FUNCTION TryConvert_BYTE_TO_WORD : BOOL
VAR_INPUT
	in : BYTE;
	out : REFERENCE TO WORD;
END_VAR

out := BYTE_TO_WORD(in);
TryConvert_BYTE_TO_WORD := TRUE;

END_FUNCTION

(* stored: Version 1.1.0.1, ProductVersion 3.1.4024.12
   POU TryConvert_BYTE_TO_WORD: Id {f96b26b8-9bd6-494d-887e-55a472e0a833}, SpecialFunc None *)
